Fanuc KAREL source: port_WDI.kl

PROGRAM TP
%NOLOCKGROUP
VAR
 x: BOOLEAN
BEGIN
 x = WDI[3]
END TP
